(* IEC 61131-3 sources: SRCI/RobotLibrary/Library/POUs/General/MC_RobotTask (part 5) *)

  RETURN;
  FOR _seqIdx := 0 TO AxesGroup.State.SequenceCountRecv
  DO
    // check new data to receive ?
    IF ( Telegram.RobToPlc.Sequence[_seqIdx].Header.SEQ_ACK <> AxesGroup.State.LastACK[_seqIdx])
    THEN
      // Check sequence payload > 0 ?
      IF (Telegram.RobToPlc.Sequence[_seqIdx].Header.PayloadLength > 0)
      THEN
        // Create log entry
        CreateLogMessagePara4 ( Timestamp   := SystemTime,
                                MessageType := MessageType.CMD,
                                Severity    := Severity.DEBUG,
                                MessageCode := 0,
                                MessageText := 'RecvData: ACK = {1}, received Sequence [{2}] with PayloadLength = {3}, Lifesign = {4}',
                                Para1       :=  UINT_TO_STRING(Telegram.RobToPlc.Sequence[_seqIdx].Header.SEQ_ACK),
                                Para2       :=  DINT_TO_STRING(_seqIdx),
                                Para3       :=  UINT_TO_STRING(Telegram.RobToPlc.Sequence[_seqIdx].Header.PayloadLength),
                                Para4       :=  BYTE_TO_STRING(Telegram.RobToPlc.Header.LifeSign));

        FOR _fragIdx := 0 TO AxesGroup.State.FragmentCountRecv[_seqIdx]
        DO
          // Check fragment payload > 0 ?
          IF (Telegram.RobToPlc.Sequence[_seqIdx].Fragment[_fragIdx].Header.PayloadLength > 0)
          THEN
            // Create log entry
            CreateLogMessagePara5 ( Timestamp   := SystemTime,
                                    MessageType := MessageType.CMD,
                                    Severity    := Severity.DEBUG,
                                    MessageCode := 0,
                                    MessageText := 'RecvData: received Fragment [{1}] with PayloadLength = {2}, CmdID <{3}> , CmdState: {4}, Fragment-Action Bits: {5}',
                                    Para1       :=  DINT_TO_STRING(0), {warning 'Add seqIdx'}
                                    Para2       :=  UINT_TO_STRING              (Telegram.RobToPlc.Sequence[_seqIdx].Fragment[_fragIdx].Header.PayloadLength),
                                    Para3       :=  DINT_TO_STRING              (Telegram.RobToPlc.Sequence[_seqIdx].Fragment[_fragIdx].Header.CmdID),
                                    Para4       :=  CMD_MESSAGE_STATE_TO_STRING (Telegram.RobToPlc.Sequence[_seqIdx].Fragment[_fragIdx].Command.Header.State),
                                    Para5       :=    FRAGMENT_ACTION_TO_STRING (Telegram.RobToPlc.Sequence[_seqIdx].Fragment[_fragIdx].Header.FragmentAction));
          END_IF
        END_FOR
      END_IF
    END_IF
  END_FOR

END_METHOD

METHOD PRIVATE ParseRecvPayloadSequence
VAR_IN_OUT
  /// Robot assignment of function
  AxesGroup        : AxesGroup;
END_VAR

VAR
  /// internal index
 _idx              : DINT;
  /// index for sequence
 _seqIdx           : DINT;
  /// index for fragment
 _fragIdx          : DINT;
  /// Amount of sequences
 _seqCount         : DINT;
  /// current payload pointer of the current sequence
 _seqPayloadPtr    : UINT;
END_VAR

  // Check 2nd sequence active ?
  IF ( _parCfg.Com.TwoSequences )
  THEN
   _seqCount := _seqCount + 1;
  END_IF

  FOR _seqIdx := 0 TO _seqCount
  DO
    // Check 2nd sequence ? -> goto 2nd sequence payload address
    IF ( _seqIdx = SECONDARY_SEQUENCE )
    THEN
      RecvData.PayloadPtr := CalculateSequencePayloadStartAdr(AxesGroup := AxesGroup,
                                                              Direction := ComDirection.ROB_TO_PLC,
                                                              Sequence  := SequenceFlag.SECONDARY_SEQUENCE);
  	END_IF

    // parste sequence header
    Telegram.RobToPlc.Sequence[_seqIdx].Header.SEQ_ACK       := RecvData.GetUint();
    Telegram.RobToPlc.Sequence[_seqIdx].Header.PayloadLength := RecvData.GetUint();

    // check new data available ?
    IF ( Telegram.RobToPlc.Sequence[_seqIdx].Header.SEQ_ACK <> AxesGroup.State.LastACK[_seqIdx])
    THEN
      // Check sequence payload available ?
      IF (Telegram.RobToPlc.Sequence[_seqIdx].Header.PayloadLength > 0)
      THEN
        // Check sequence payload length is valid ?
        IF ( Telegram.RobToPlc.Sequence[_seqIdx].Header.PayloadLength > _parCfg.Com.TelegramLengthRobToPlc )
        THEN
          // Create log entry for payload not valid
          CreateLogMessagePara2 ( Timestamp   := SystemTime,
                                  MessageType := MessageType.CMD,
                                  Severity    := Severity.DEBUG,
                                  MessageCode := 0,
                                  MessageText := 'Invalid sequence payload length, Sequence = {1}, PayloadLength = {2} ',
                                  Para1       :=  DINT_TO_STRING(_seqIdx),
                                  Para2       :=  UINT_TO_STRING(Telegram.RobToPlc.Sequence[_seqIdx].Header.PayloadLength));
                                  RETURN;
        ELSE
          // Create log entry
          CreateLogMessagePara4 ( Timestamp   := SystemTime,
                                  MessageType := MessageType.CMD,
                                  Severity    := Severity.DEBUG,
                                  MessageCode := 0,
                                  MessageText := 'RecvData: ACK = {1}, received Sequence [{2}] with PayloadLength = {3}, Lifesign = {4}',
                                  Para1       :=  UINT_TO_STRING(Telegram.RobToPlc.Sequence[_seqIdx].Header.SEQ_ACK),
                                  Para2       :=  DINT_TO_STRING(_seqIdx),
                                  Para3       :=  UINT_TO_STRING(Telegram.RobToPlc.Sequence[_seqIdx].Header.PayloadLength),
                                  Para4       :=  BYTE_TO_STRING(Telegram.RobToPlc.Header.LifeSign));
        END_IF

        // processing sequence payload
        WHILE ( _seqPayloadPtr < Telegram.RobToPlc.Sequence[_seqIdx].Header.PayloadLength )
        DO
          // parse header
          Telegram.RobToPlc.Sequence[_seqIdx].Fragment[_fragIdx].Header.CmdID          := RecvData.GetUint();
          Telegram.RobToPlc.Sequence[_seqIdx].Fragment[_fragIdx].Header.Reserve        := RecvData.GetByte();
          Telegram.RobToPlc.Sequence[_seqIdx].Fragment[_fragIdx].Header.FragmentAction := RecvData.GetByte();
          Telegram.RobToPlc.Sequence[_seqIdx].Fragment[_fragIdx].Header.PayloadPointer := RecvData.GetUint();
          Telegram.RobToPlc.Sequence[_seqIdx].Fragment[_fragIdx].Header.PayloadLength  := RecvData.GetUint();

          // add header size to payload pointer
         _seqPayloadPtr := _seqPayloadPtr + SIZEOF(Telegram.RobToPlc.Sequence[_seqIdx].Fragment[_fragIdx].Header);

          // Check fragment payload available ?
          IF (Telegram.RobToPlc.Sequence[_seqIdx].Fragment[_fragIdx].Header.PayloadLength > 0)
          THEN
            // Check fragment payload length is valid ?
            IF ( Telegram.RobToPlc.Sequence[_seqIdx].Fragment[_fragIdx].Header.PayloadLength > _parCfg.Com.TelegramLengthRobToPlc )
            THEN
              // Create log entry for payload not valid
              CreateLogMessagePara2 ( Timestamp   := SystemTime,
                                      MessageType := MessageType.CMD,
                                      Severity    := Severity.DEBUG,
                                      MessageCode := 0,
                                      MessageText := 'Invalid fragment payload length, Sequence = {1}, PayloadLength = {2} ',
                                      Para1       :=  DINT_TO_STRING(_seqIdx),
                                      Para2       :=  UINT_TO_STRING(Telegram.RobToPlc.Sequence[_seqIdx].Fragment[_fragIdx].Header.PayloadLength));
                                      RETURN;
            END_IF

            // Fill Response payload
            FOR _idx := Telegram.RobToPlc.Sequence[_seqIdx].Fragment[_fragIdx].Header.PayloadPointer TO Telegram.RobToPlc.Sequence[_seqIdx].Fragment[_fragIdx].Header.PayloadLength -1
            DO
              Telegram.RobToPlc.Sequence[_seqIdx].Fragment[_fragIdx].Command.Payload[_idx] := RecvData.GetByte();
              // inc payload pointer
             _seqPayloadPtr := _seqPayloadPtr + SIZEOF(BYTE);
            END_FOR

            // Add Response to ACR
            AxesGroup.Acyclic.ActiveCommandRegister.AddRsp(Telegram.RobToPlc.Sequence[_seqIdx].Fragment[_fragIdx]);

            // Only for debugging - header is part of the payload itself
            Telegram.RobToPlc.Sequence[_seqIdx].Fragment[_fragIdx].Command.Header.State                 :=      GetHalfeByteLo( Value :=  Telegram.RobToPlc.Sequence[_seqIdx].Fragment[_fragIdx].Command.Payload[0]);
            Telegram.RobToPlc.Sequence[_seqIdx].Fragment[_fragIdx].Command.Header.ParSeq                :=      GetHalfeByteHi( Value :=  Telegram.RobToPlc.Sequence[_seqIdx].Fragment[_fragIdx].Command.Payload[0]);
            Telegram.RobToPlc.Sequence[_seqIdx].Fragment[_fragIdx].Command.Header.AlarmMessageSeverity  :=        BYTE_TO_SINT(           Telegram.RobToPlc.Sequence[_seqIdx].Fragment[_fragIdx].Command.Payload[1]);
            Telegram.RobToPlc.Sequence[_seqIdx].Fragment[_fragIdx].Command.Header.AlarmMessageCode      :=  CombineBytesToUint( HiByte := Telegram.RobToPlc.Sequence[_seqIdx].Fragment[_fragIdx].Command.Payload[2],
                                                                                                                                LoByte := Telegram.RobToPlc.Sequence[_seqIdx].Fragment[_fragIdx].Command.Payload[3]);
            // Create log entry
            CreateLogMessagePara5 ( Timestamp   := SystemTime,
                                    MessageType := MessageType.CMD,
                                    Severity    := Severity.DEBUG,
                                    MessageCode := 0,
                                    MessageText := 'RecvData: received Fragment [{1}] with PayloadLength = {2}, CmdID <{3}> , CmdState: {4}, Fragment-Action Bits: {5}',
                                    Para1       :=  DINT_TO_STRING(_seqIdx),
                                    Para2       :=  UINT_TO_STRING              (Telegram.RobToPlc.Sequence[_seqIdx].Fragment[_fragIdx].Header.PayloadLength),
                                    Para3       :=  DINT_TO_STRING              (Telegram.RobToPlc.Sequence[_seqIdx].Fragment[_fragIdx].Header.CmdID),
                                    Para4       :=  CMD_MESSAGE_STATE_TO_STRING (Telegram.RobToPlc.Sequence[_seqIdx].Fragment[_fragIdx].Command.Header.State),
                                    Para5       :=    FRAGMENT_ACTION_TO_STRING (Telegram.RobToPlc.Sequence[_seqIdx].Fragment[_fragIdx].Header.FragmentAction));
          END_IF

          // Check still payload left ? -> goto next fragment
          IF ( _seqPayloadPtr < Telegram.RobToPlc.Sequence[_seqIdx].Header.PayloadLength )
          THEN
           _fragIdx := _fragIdx + 1;
          END_IF

          // Check fragment index limit reached ?
          IF ( _fragIdx > RobotLibraryParameter.FRAGMENT_MAX )
          THEN
            // Create log entry
            CreateLogMessagePara1 ( Timestamp   := SystemTime,
                                    MessageType := MessageType.CMD,
                                    Severity    := Severity.DEBUG,
                                    MessageCode := 0,
                                    MessageText := 'Fragment index out of range, _fragIdx = {1} ',
                                    Para1       :=  DINT_TO_STRING(_fragIdx));
                                    RETURN;
          END_IF
        END_WHILE
      END_IF
    END_IF
  END_FOR

END_METHOD

METHOD Reset
VAR_IN_OUT
  /// Robot assignment of function
  AxesGroup : AxesGroup;
END_VAR

  // reset flags
  Busy              := FALSE;
  Initialized       := FALSE;
  Synchronized      := FALSE;
  Error             := FALSE;
  ErrorID           := 0;
  ErrorAddTxt       := '';
  WarningID         := 0;
  InfoID            := 0;

  // Reset internal functon blocks
  _exchangeConfiguration      .Enable  := FALSE;
  _readRobotData              .Execute := FALSE;
  _readMessages               .Enable  := FALSE;
  _readToolData               .Execute := FALSE;
  _readFrameData              .Execute := FALSE;
  _readLoadData               .Execute := FALSE;
  _readWorkArea               .Execute := FALSE;
  _readRobotSWLimits          .Execute := FALSE;
  _readRobotDefaultDynamics   .Execute := FALSE;
  _readRobotReferenceDynamics .Execute := FALSE;
  _writeToolData              .Execute := FALSE;
  _writeFrameData             .Execute := FALSE;
  _writeLoadData              .Execute := FALSE;
  _writeWorkArea              .Execute := FALSE;
  _writeRobotSWLimits         .Execute := FALSE;
  _writeRobotDefaultDynamics  .Execute := FALSE;
  _writeRobotReferenceDynamics.Execute := FALSE;

  // Set Client error to force server error
  AxesGroup.Cyclic.PlcToRob.Control := ControlHalfByte.NONE;

  // Reset synchronisation state variables
  AxesGroup.State.SyncStatePlc.InSync.Frame             := FALSE;
  AxesGroup.State.SyncStatePlc.InSync.Tool              := FALSE;
  AxesGroup.State.SyncStatePlc.InSync.Load              := FALSE;
  AxesGroup.State.SyncStatePlc.InSync.WorkArea          := FALSE;
  AxesGroup.State.SyncStatePlc.InSync.SwLimits          := FALSE;
  AxesGroup.State.SyncStatePlc.InSync.DefaultDynamics   := FALSE;
  AxesGroup.State.SyncStatePlc.InSync.ReferenceDynamics := FALSE;

  AxesGroup.State.SyncStatePlc.UnSyncNo.Frame    := 0;
  AxesGroup.State.SyncStatePlc.UnSyncNo.Tool     := 0;
  AxesGroup.State.SyncStatePlc.UnSyncNo.Load     := 0;
  AxesGroup.State.SyncStatePlc.UnSyncNo.WorkArea := 0;

  AxesGroup.State.SyncStateRc .InSync.Frame             := FALSE;
  AxesGroup.State.SyncStateRc .InSync.Tool              := FALSE;
  AxesGroup.State.SyncStateRc .InSync.Load              := FALSE;
  AxesGroup.State.SyncStateRc .InSync.WorkArea          := FALSE;
  AxesGroup.State.SyncStateRc .InSync.SwLimits          := FALSE;
  AxesGroup.State.SyncStateRc .InSync.DefaultDynamics   := FALSE;
  AxesGroup.State.SyncStateRc .InSync.ReferenceDynamics := FALSE;

  AxesGroup.State.SyncStateRc .UnSyncNo.Frame    := 0;
  AxesGroup.State.SyncStateRc .UnSyncNo.Tool     := 0;
  AxesGroup.State.SyncStateRc .UnSyncNo.Load     := 0;
  AxesGroup.State.SyncStateRc .UnSyncNo.WorkArea := 0;

  // Reset active command register
  AxesGroup.Acyclic.ActiveCommandRegister.Reset();

  // reset step counters
  _stepCmd                   := 0;
  _stepSyncFrameData         := 0;
  _stepSyncLoadData          := 0;
  _stepSyncDefaultDynamics   := 0;
  _stepSyncReferenceDynamics := 0;
  _stepSyncSWLimits          := 0;
  _stepSyncToolData          := 0;
  _stepSyncWorkArea          := 0;

END_METHOD
